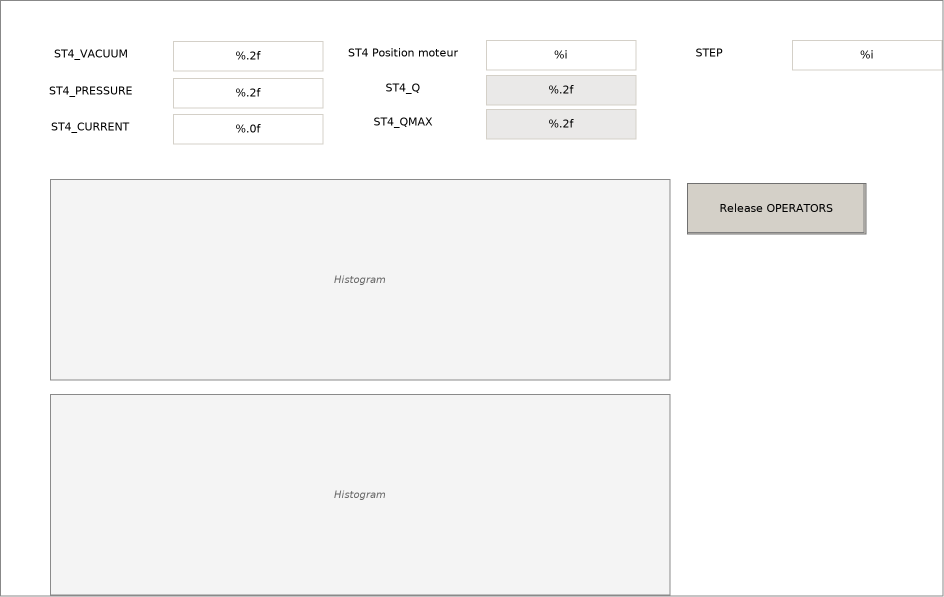
VISUALIZATION ST4  // 944x597
    Textfield (173,41 150x30), "%.2f", text variable: ST4_VACUUM
    Label (16,39 150x30), "ST4_VACUUM"
    Textfield (173,78 150x30), "%.2f", text variable: ST4_PRESSURE
    Label (16,76 150x30), "ST4_PRESSURE"
    Textfield (173,114 150x30), "%.0f", text variable: ST4_COURANT
    Label (15,112 150x30), "ST4_CURRENT"
    Textfield (486,40 150x30), "%i", text variable: Flag_Variables.FLAGS.MOTOR_ST4_ACTUAL_POSITION
    Label (328,38 150x30), "ST4 Position moteur"
    Textfield (486,75 150x30), "%.2f", text variable: ST4_Q
    Label (328,73 150x30), "ST4_Q"
    Textfield (486,109 150x30), "%.2f", text variable: ST4_QMAX
    Label (328,107 150x30), "ST4_QMAX"
    Histogram (50,179 620x201), scale format: %.1f, scale 20..30
        p1518820177: Flag_Variables.QMAX_ARRAY
        p102497268: Flag_Variables.QMAX_ARRAY
        p788070771: ARRAY [1..50] OF REAL
    Histogram (50,394 620x201), scale format: %.1f, scale 10..20
        p1518820177: Flag_Variables.Q_ARRAY
        p102497268: Flag_Variables.Q_ARRAY
        p788070771: ARRAY [1..50] OF REAL
    Button (687,183 179x51), "Release OPERATORS"
        tap Flag_Variables.FLAGS.DEBUG_OPERATOR
    Label (634,38 150x30), "STEP"
    Textfield (792,40 150x30), "%i", text variable: IOs_Variables.PROG_STEPS.ST4
END_VISUALIZATION

(* stored: Version 1.1.0.1, ProductVersion 3.1.0.26
   Visu ST4: Id {dc7ff86e-8f16-40cc-be83-31719ff335a5} *)
